FUNCTION UINT_TO_SIZE : ST_SIZE
VAR_INPUT
	nValue : UINT;
END_VAR

UINT_TO_SIZE.nValue := nValue;

END_FUNCTION

(* stored: Version 1.1.0.1, ProductVersion 3.1.4024.15
   POU UINT_TO_SIZE: Id {1e36d644-d847-4e21-8285-fe5478178171}, SpecialFunc None *)
